// TIA Portal project "Project2" (V15.1)

(* hardware
DEVICE "S7-1200 station_1"  S7-1200 Station
   slot 0: "Rack_0"  S7-1200 Rack  Rack  V1.0
   slot 1: "PLC_1"  CPU 1211C DC/DC/Rly  6ES7 211-1HD30-0XB0  V2.2
*)

// ===== PLC "PLC_1"  CPU 1211C DC/DC/Rly =====

VAR_GLOBAL   // PLC tag table "Default tag table"
   "STOP" AT %I0.0 : Bool;
   "İleriStart" AT %I0.1 : Bool;
   "GeriStart" AT %I0.2 : Bool;
   "İleriKont" AT %I0.3 : Bool;
   "GeriKont" AT %I0.4 : Bool;
   "StopLamba" AT %I0.5 : Bool;
END_VAR

ORGANIZATION_BLOCK "Main"   // OB1, LAD, ProgramCycle
TITLE = "Main Program Sweep (Cycle)"
{ S7_Optimized_Access := 'TRUE' }
VERSION : 0.1
BEGIN

REGION Network 1
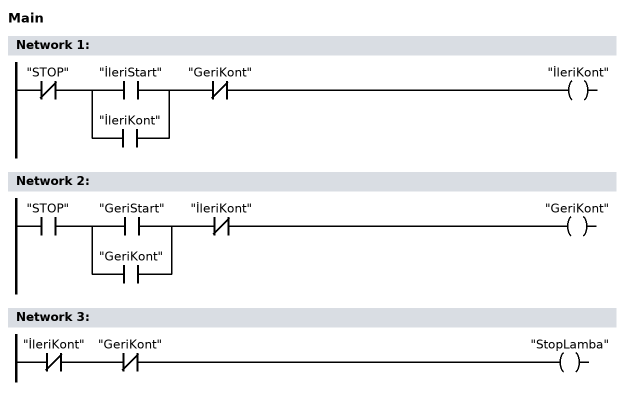
   RUNG wire#powerrail
      I_Contact( "STOP" )
      wire#w1
      Contact( "İleriStart" )
      wire#w2
      I_Contact( "GeriKont" )
      Coil( "İleriKont" )
   END_RUNG
   RUNG wire#w1
      Contact( "İleriKont" )
   END_RUNG wire#w2
   RUNG wire#powerrail
   END_RUNG
   // the same network as SCL:
   "İleriKont" := NOT "STOP" AND ("İleriStart" OR "İleriKont") AND NOT "GeriKont";
END_REGION

REGION Network 2
   RUNG wire#powerrail
      Contact( "STOP" )
      wire#w1
      Contact( "GeriStart" )
      wire#w2
      I_Contact( "İleriKont" )
      Coil( "GeriKont" )
   END_RUNG
   RUNG wire#w1
      Contact( "GeriKont" )
   END_RUNG wire#w2
   // the same network as SCL:
   "GeriKont" := "STOP" AND ("GeriStart" OR "GeriKont") AND NOT "İleriKont";
END_REGION

REGION Network 3
   RUNG wire#powerrail
      I_Contact( "İleriKont" )
      I_Contact( "GeriKont" )
      Coil( "StopLamba" )
   END_RUNG
   // the same network as SCL:
   "StopLamba" := NOT "İleriKont" AND NOT "GeriKont";
END_REGION
END_ORGANIZATION_BLOCK